PROGRAM MAIN
VAR
END_VAR

END_PROGRAM

(* stored: Version 1.1.0.1
   POU MAIN: Id {99b7bca1-6f1d-4e64-9b5c-cc4d83d7cd89} *)
